{attribute addProperty BoxType "EL1859-0000-0016"}
{attribute addProperty Id "ChannelAT %I*ARRAY[0..7] OF Channel_E4AEF59E6480Channel_1AT %Q*ARRAY[0..7] OF Channel_7F374EB06480WcStateAT %I*WcState_98A4DF7520.250InfoDataAT %I*InfoData_192954DE1620"}
{attribute addProperty CRC "4038043443"}
{attribute addProperty SizeInBites "146"}
{attribute addProperty SizeInBytes "18.25"}
TYPE EL1859_538B459D :
STRUCT
	{attribute addProperty Name "Channel"}
	Channel : ARRAY[0..7] OF Channel_E4AEF59E;
	{attribute addProperty Name "Channel_1"}
	Channel_1 : ARRAY[0..7] OF Channel_7F374EB0;
	{attribute addProperty Name "WcState"}
	WcState : WcState_98A4DF75;
	{attribute addProperty Name "InfoData"}
	InfoData : InfoData_192954DE;
END_STRUCT
END_TYPE

(* stored: Version 1.2.0.0, ProductVersion 3.1.4024.9
   DUT EL1859_538B459D: Id {f7cb0cc4-918c-40c4-b1e5-6c8119826536} *)
